TYPE aT_Motor :
STRUCT
	SetSpeed: LREAL;
	Speed: LREAL;
END_STRUCT
END_TYPE

(* stored: Version 1.1.0.1, ProductVersion 3.1.4024.4
   DUT aT_Motor: Id {3d418655-d2fb-4fbe-a40b-73514e89641a} *)
